{attribute 'qualified_only'}
VAR_GLOBAL
	Axis1 : AXIS_REF;
END_VAR

(* stored: Version 1.1.0.1, ProductVersion 3.1.4024.13
   GVL Axes: Id {2f45a541-0c5f-4bea-b434-313df9ffab21} *)
